(* CODESYS project FBD1-bad_engineering.project

Project tree, tasks and I/O mapping:
  Device : CODESYS Control Win V3, 3S - Smart Software Solutions GmbH, order no. 305021, version 3.5.10.30
    application Application
      libraries: Standard, * (System)
      task MainTask (cyclic, interval t#20ms, priority 1) calls PLC_PRG
      task VISU_TASK (cyclic, interval 100 ms, priority 31) calls VisuElems.Visu_Prg
      program PLC_PRG [FBD]
      visualisation Visualization
  text list GlobalTextList
*)

// Device/Application/PLC_PRG
PROGRAM PLC_PRG
VAR
	CTU_1: CTU;
	PV1: WORD := 3;
	Value: WORD;
	Contact1: BOOL;
END_VAR

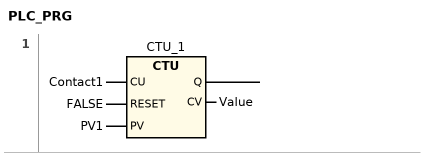
// NETWORK 1
CTU_1(CU := Contact1, RESET := FALSE, PV := PV1, CV => Value); // CTU

END_PROGRAM

// Device/Application/Visualization
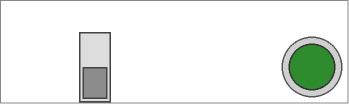
VISUALIZATION Visualization  // 349x104
    DipSwitch (60,32 70x70), variable: PLC_PRG.Contact1, behaviour: TOGGLE, style: Switch-DipSwitch-Gray
    Lamp1 (277,32 70x70), variable: PLC_PRG.CTU_0.Q, style: Lamp-Lamp1-Green
END_VISUALIZATION
